Fanuc KAREL source: IO0023.KL

-- PROVISIONAL review KL for V770-1; original PC SHA256 4b5c32718254d7945f7ec9d5aa11934edc2b70bc507377cd055a7ef227adaec8
-- Incomplete behavior may be omitted. Consult companion uncertainty JSON. Do not deploy.
PROGRAM IO0023
%NOLOCKGROUP
-- UNRESOLVED_LOCAL_POOL 5 cells at code offset 13; source declarations unknown
-- DIRECT_LOCAL_WORD_ACCESS alone does not prove INTEGER, REAL, or BOOLEAN
BEGIN
  -- UNRESOLVED_PC offsets 0-18; opcodes 2B,2C,7B
  -- UNRESOLVED_PC offsets 23-30; opcodes 9D,23
  -- UNRESOLVED_PC offsets 35-49; opcodes 2E,22,9D,33,35
  -- UNRESOLVED_PC offsets 54-61; opcodes 9D,23
  -- UNRESOLVED_PC offsets 66-77; opcodes 2E,23
  -- UNRESOLVED_PC offsets 82-90; opcodes 9D,2E,1A
  -- UNRESOLVED_PC offsets 95-99; opcodes 7F
  -- UNRESOLVED_PC offsets 104-108; opcodes 27,AA
  -- UNRESOLVED_PC offsets 113-117; opcodes 7F
END IO0023
